(*This function block (FB) is resposible for handling the set method calls. It provides the following void methods; 
buttonPlayPause, buttonStickMinus, buttonStickPlus, buttonStop, changeProjectSpeed, moveRelativePTP, setJointsPTP. *)
FUNCTION_BLOCK FB_HandleSetTM
VAR_INPUT
END_VAR
VAR_OUTPUT
END_VAR
VAR
	//stRobotArmObjectTM : ST_RobotArmObjectTM;
	
	//Initialize function block
	{attribute 'OPC.UA.DA':='0'}
	fbModbusWriteTM : FB_ModbusWriteTM;
	
	//reference object from command window
	{attribute 'OPC.UA.DA':='0'}
	stRobotArmReferenceTM : ST_RobotArmObjectTM;
END_VAR



(*--------------- Allow access from command window if requested---------------*)
IF GVL_CommandWindow.bCmdMoveRelPTP OR GVL_CommandWindow.bCmdMoveRelLinear THEN
	IF GVL_CommandWindow.bCmdMoveRelPTP THEN
		GVL_CommandWindow.bCmdMoveRelPTP := FALSE;
		stRobotArmReferenceTM.cmdID := 1;
	END_IF
	IF GVL_CommandWindow.bCmdMoveRelLinear THEN
		GVL_CommandWindow.bCmdMoveRelLinear := FALSE;
		stRobotArmReferenceTM.cmdID := 2;
	END_IF
	
	stRobotArmReferenceTM.fX := GVL_CommandWindow.fX_Ref;
	stRobotArmReferenceTM.fY := GVL_CommandWindow.fY_Ref;
	stRobotArmReferenceTM.fZ := GVL_CommandWindow.fZ_Ref;
	stRobotArmReferenceTM.fRX := GVL_CommandWindow.fRX_Ref;
	stRobotArmReferenceTM.fRY := GVL_CommandWindow.fRY_Ref;
	stRobotArmReferenceTM.fRZ := GVL_CommandWindow.fRZ_Ref;
	fbModbusWriteTM(stReferenceTM := stRobotArmReferenceTM);
END_IF

IF GVL_CommandWindow.bCmdSetJointsPTP THEN
	GVL_CommandWindow.bCmdSetJointsPTP := FALSE;
	stRobotArmReferenceTM.cmdID := 3;
	stRobotArmReferenceTM.fTheta1 := GVL_CommandWindow.fTheta1_Ref;
	stRobotArmReferenceTM.fTheta2 := GVL_CommandWindow.fTheta2_Ref;
	stRobotArmReferenceTM.fTheta3 := GVL_CommandWindow.fTheta3_Ref;
	stRobotArmReferenceTM.fTheta4 := GVL_CommandWindow.fTheta4_Ref;
	stRobotArmReferenceTM.fTheta5 := GVL_CommandWindow.fTheta5_Ref;
	stRobotArmReferenceTM.fTheta6 := GVL_CommandWindow.fTheta6_Ref;
	fbModbusWriteTM(stReferenceTM := stRobotArmReferenceTM);
END_IF


(*--------------- TO DO: Return the answer for class methods, external access---------------*)

// Press the Play/Pause button of the robot stick
{attribute 'TcRpcEnable':='1'}
METHOD buttonPlayPause : BOOL // FALSE: finished
VAR_INPUT
END_VAR
fbModbusWriteTM.writeSingleCoil(nMBAddr5 := 16#1BC0); //starting modbus client with address 7104 (Play/Pause)

buttonPlayPause := FALSE;  //indicates that the job of the function is finished
END_METHOD

// Press the Minus(-) button of the robot stick 
{attribute 'TcRpcEnable':='1'}
METHOD buttonStickMinus : BOOL // FALSE: finished
VAR_INPUT
END_VAR

fbModbusWriteTM.writeSingleCoil(nMBAddr5 := 16#1BC3); //starting modbus client with address 7107 (Stick-)

buttonStickMinus := FALSE;  //indicates that the job of the function is finished
END_METHOD

// Press the Plus(+) button of the robot stick
{attribute 'TcRpcEnable':='1'}
METHOD buttonStickPlus : BOOL // FALSE: finished
VAR_INPUT
END_VAR

fbModbusWriteTM.writeSingleCoil(nMBAddr5 := 16#1BC2); //starting modbus client with address 7106 (Stick+)

buttonStickPlus := FALSE;  //indicates that the job of the function is finished
END_METHOD

// Press the Stop button of the robot stick
{attribute 'TcRpcEnable':='1'}
METHOD buttonStop : BOOL // FALSE: finished
VAR_INPUT
END_VAR


fbModbusWriteTM.writeSingleCoil(nMBAddr5 := 16#1BC1); //starting modbus client with address 7105 (Stop)

buttonStop := FALSE; //indicates that the job of the function is finished
END_METHOD

// Change the project in range 0% to 100%
{attribute 'TcRpcEnable':='1'}
METHOD changeProjectSpeed : INT // FALSE: finished
VAR_INPUT
	projectSpeed : INT; //Project speed (multiples of 5)
END_VAR
VAR
	nValueInt : WORD;
	remainder : INT;
END_VAR
IF projectSpeed < 5 THEN
	projectSpeed := 5; //min 5%
ELSIF projectSpeed > 100 THEN
	projectSpeed := 100; //max 10%
END_IF

remainder := projectSpeed MOD 5;
projectSpeed := projectSpeed - remainder; //only multiples of 5 
nValueInt := INT_TO_WORD(projectSpeed);


fbModbusWriteTM.writeSingleRegister(nMBAddr6 := 16#1BBD,nValue6 := nValueInt); //starting modbus client with address 7101 (Change Project Speed)

changeProjectSpeed := 2;  //indicates that the job of the function is finished
END_METHOD

//Move the robot point-to-point(PTP) in relative cartesian coordinate frame
{attribute 'TcRpcEnable':='1'}
METHOD moveRelativePTP : BOOL // FALSE: finished
VAR_INPUT
	fX : REAL := 0; // Translation in the x-axis
	fY : REAL := 0; // Translation in the y-axis
	fZ : REAL := 0; // Translation in the z-axis
	fRX : REAL := 0; // Rotation in the x-axis
	fRY : REAL := 0; // Rotation in the y-axis
	fRZ : REAL := 0; // Rotation in the z-axis
END_VAR
VAR
	stRobotArmRefTM : ST_RobotArmObjectTM;
END_VAR
stRobotArmRefTM.cmdID := MoveCartesianPTP;
stRobotArmRefTM.fX := fX;
stRobotArmRefTM.fY := fY;
stRobotArmRefTM.fZ := fZ;
stRobotArmRefTM.fRX := fRX;
stRobotArmRefTM.fRY := fRY;
stRobotArmRefTM.fRZ := fRZ;

fbModbusWriteTM(stReferenceTM := stRobotArmRefTM); //start Modbus TCP Client 

moveRelativePTP := FALSE;  //indicates that the job of the function is finished
END_METHOD

// Move the robot joints point-to-point(PTP)
{attribute 'TcRpcEnable':='1'}
METHOD setJointsPTP : BOOL // FALSE: finished
VAR_INPUT
	fTheta1 : REAL := 0; // Joint 1
	fTheta2 : REAL := 0; // Joint 2
	fTheta3 : REAL := 0; // Joint 3
	fTheta4 : REAL := 0; // Joint 4
	fTheta5 : REAL := 0; // Joint 5 
	fTheta6 : REAL := 0; // Joint 6
END_VAR
VAR
	stRobotArmRefTM : ST_RobotArmObjectTM;
END_VAR
stRobotArmRefTM.cmdID := SetJointPositions;
stRobotArmRefTM.fTheta1 := fTheta1;
stRobotArmRefTM.fTheta2 := fTheta2;
stRobotArmRefTM.fTheta3 := fTheta3;
stRobotArmRefTM.fTheta4 := fTheta4;
stRobotArmRefTM.fTheta5 := fTheta5;
stRobotArmRefTM.fTheta6 := fTheta6;

fbModbusWriteTM(stReferenceTM:= stRobotArmRefTM); //start Modbus TCP Client 

setJointsPTP := FALSE;  //indicates that the job of the function is finished
END_METHOD

END_FUNCTION_BLOCK

(* stored: Version 1.1.0.1, ProductVersion 3.1.4024.11
   POU FB_HandleSetTM: Id {6d8cf4ea-1acf-46ca-b535-92c6f38dbe51}, SpecialFunc None
   Method buttonPlayPause: Id {0b1d57f9-a4b5-44da-b5b5-20ff9edd9e1a}
   Method buttonStickMinus: Id {629aaa79-b467-4617-a0d7-2104da3bed0d}
   Method buttonStickPlus: Id {ccad1382-771e-438e-a5ba-0fa6fb7df5c8}
   Method buttonStop: Id {87a8389f-2227-49a5-98c8-0ace10da4a71}
   Method changeProjectSpeed: Id {e0973733-aa90-49c8-b87e-f3a4990b0108}
   Method moveRelativePTP: Id {ce9a3435-a40a-4dd1-b1c9-e59b41424958}
   Method setJointsPTP: Id {86b01414-8c9d-4d34-80ad-9ec44c360771} *)
